FUNCTION_BLOCK Test_TExecutionWhenReady_Start_SelectsStarting EXTENDS T_UnitTestbase
VAR
    Execution : T_Execution;
END_VAR

METHOD Init
// Setup...
Execution.FB_init(bInitRetains := FALSE,
                  bInCopyCode  := FALSE);
END_METHOD

{attribute 'analysis' := '-33'} // inhibit unused variable warning
METHOD RunTest
VAR_OUTPUT
    TestCompleted : BOOL;
    TestFailed    : BOOL;
END_VAR
// Test...
Execution.Start();

TestFailed S= NOT AssertTrue(Source    := TestName,
                             Condition := Execution.Starting,
                             Message   := 'Execution.Starting not true');

TestCompleted := TRUE;
END_METHOD

END_FUNCTION_BLOCK

(* stored: Version 1.1.0.1, ProductVersion 3.1.4024.12
   POU Test_TExecutionWhenReady_Start_SelectsStarting: Id {0349ca1d-2308-406f-93fd-15ff4a011555}, SpecialFunc None
   Method Init: Id {a400d995-282b-47a4-88aa-7ef559a0d3a3}
   Method RunTest: Id {f67e2ae3-dccd-435c-ab38-3d5cd2aad280} *)
